{attribute 'qualified_only'}
{attribute 'strict'}
TYPE E_HomingRoutines :
(
    eNoHoming := 0,

    //0X: LIMIT Switch
    //Home to bBwdLimit, record position on first approach
    eHomeToLimit_Bwd := 1,
    //Home to bFwdLimit, record position on first approach
    eHomeToLimit_Fwd := 2,
    //Find bBwdLimit (using towardsCam speed), then reverse direction looking FOR falling edge (using fromCam speed)
    //eHomeToLimit_Bwd_2Speeds := 3,
    //Find bFwdLimit (using towardsCam speed), then reverse direction looking for falling edge (using fromCam speed)
    //eHomeToLimit_Fwd_2Speeds := 4,

    //1X: Home Sensor
    //Home to bHome in Bwd direction (will reverse direction if limit hit), record position on first approach
    eHomeToRef_Bwd := 11,
    //Home to bHome in Fwd direction (will reverse direction if limit hit), record position on first approach
    eHomeToRef_Fwd := 12,
    //Find bHome in Bwd direction (using towardsCam speed) then reverse direction looking for falling edge (using fromCam speed), will reverse direction if limit hit
    //eHomeToRef_Bwd_2Speeds := 13,
    //Find bHome in Fwd direction (using towardsCam speed) then reverse direction looking for falling edge (using fromCam speed), will reverse direction if limit hit
    //eHomeToRef_Fwd_2Speeds := 14,

    //2X: Enc Pulse
    //Home to EncRefPulse in Bwd direction (used for single turn rotary axis without limit switches)
    eHomeToEncPulse_Bwd := 21,
    //Home to EncRefPulse in Fwd direction (used for single turn rotary axis without limit switches)
    eHomeToEncPulse_Fwd := 22,
    //Home to EncRefPulse via bBwdLimit (using towardsCam speed), then reverse direction looking for falling edge on ref pulse (using fromCam speed)
    eHomeToEncPulse_viaBwdLimit := 23,
    //Home to EncRefPulse via bFwdLimit (using towardsCam speed), then reverse direction looking for falling edge on ref pulse (using fromCam speed)
    eHomeToEncPulse_viaFwdLimit := 24,

    //3X: Home To Mechanical Block (Lag based StepBlockDetection)
    //Home towards a mechanical block in Bwd direction
    eHomeToBlock_Bwd := 30,
    //Home towards a mechanical block in Fwd direction
    eHomeToBlock_Fwd := 31,

    //9X: Software
    eHomeDirect := 90 //Set position directly to fHomePosition
) := eHomeDirect;
END_TYPE

(* stored: Version 1.1.0.1, ProductVersion 3.1.4024.12
   EnumerationTextList E_HomingRoutines: Id {80602f9f-a7d4-4c82-a41f-735a98acfb74} *)
